{attribute 'no_explicit_call' := 'do not call this FB directly'}{attribute 'enable_dynamic_creation'}
FUNCTION_BLOCK FINAL IntDisplayNode EXTENDS Node
VAR
	in : _INT(0);
	display : _INT(0);
END_VAR

METHOD PUBLIC Clone : I_Node
VAR
	pNode : POINTER TO IntDisplayNode;
END_VAR
pNode := __NEW(IntDisplayNode);
Clone := pNode^;
END_METHOD

METHOD FB_init : BOOL
VAR_INPUT
	bInitRetains : BOOL; // if TRUE, the retain variables are initialized (warm start / cold start)
	bInCopyCode : BOOL;  // if TRUE, the instance afterwards gets moved into the copy code (online change)
END_VAR
AddInput('in', in);
AddContent('display', display);
END_METHOD

METHOD PROTECTED OnExecute : HRESULT
display.Value := in.Value;
END_METHOD

END_FUNCTION_BLOCK

(* stored: Version 1.1.0.1, ProductVersion 3.1.4024.12
   POU IntDisplayNode: Id {3bd6350d-d4bd-06bc-0c94-08b70fb6859d}, SpecialFunc None
   Folder Constructor: Id {bd80cb79-538a-04cc-0cef-192708d34cd5}
   Method Clone: Id {4db5e58e-8b4f-0406-25bf-9435efb0f53a}
   Method FB_init: Id {d8cbd0df-fd6c-03fc-14da-a7d761901115}
   Method OnExecute: Id {540014d4-7c2b-0099-1eda-18753a8af52d} *)
